{attribute 'qualified_only'}
VAR_GLOBAL
	
	CoolGuyAlert : BOOL;
	DiskGolfMaster : BOOL;
	
END_VAR

(* stored: Version 1.1.0.1, ProductVersion 3.1.4024.12
   GVL GVL: Id {362ef228-ec18-4303-943c-25db6ef6ea90} *)
